FUNCTION_BLOCK DynamicStringBuffer_TEST EXTENDS FB_TestSuite
VAR_INPUT
END_VAR
VAR_OUTPUT
END_VAR
VAR
END_VAR

LogsManyMessagesForManyCycles();

METHOD LogsManyMessagesForManyCycles
VAR_INPUT
END_VAR
VAR
	result: STRING := '';
	expected: STRING := '';
	i: UDINT;
END_VAR

VAR CONSTANT
	CYCLES: UDINT := 30;
	MESSAGES: UDINT := 30;
END_VAR

VAR_INST
	cycleCount: UDINT := 0;
	LogsManyMessagesForManyCyclesLogger: TcLogCore(nBufferSize := 30*30*280); // cycles * messages * (max string length + fifo overhead (estimated))
	logger: TcLog;
END_VAR
TEST('LogsManyMessagesForManyCycles');

LogsManyMessagesForManyCyclesLogger
	.WriteToFile('c:\logs\', 'test.txt')
	.RunLogger();
logger.SetLogger(LogsManyMessagesForManyCyclesLogger);

IF cycleCount < CYCLES THEN
	FOR i:=0 TO MESSAGES DO
		logger
			.AppendString('Cycle: ')
			.AppendString(UDINT_TO_STRING(cycleCount))
			.AppendString(', Message: ')
			.AppendString(UDINT_TO_STRING(i))
			.Error('');	
	END_FOR
END_IF
cycleCount := cycleCount + 1;

// Length of operations (empirically determined):
// file open: 		2 cycles
// pop from fifo: 	1-2 cycle
// write to file: 	2 cylces
// close file:		2 cylces
// => thus for x messages you need 4 * x + 4 cycles

// Catch any occuring error message
IF LEN(LogsManyMessagesForManyCyclesLogger.Error.Info) > 0 THEN
	result := LogsManyMessagesForManyCyclesLogger.Error.Info;
END_IF

IF cycleCount > (CYCLES * MESSAGES * 4 + 10) THEN 
	AssertEquals(Expected := expected,
				 Actual := result,
				 Message := result);
 
	TEST_FINISHED();
END_IF
END_METHOD

END_FUNCTION_BLOCK

(* stored: Version 1.1.0.1, ProductVersion 3.1.4024.11
   POU DynamicStringBuffer_TEST: Id {03045c1a-5281-4fe3-bc16-4d9ce12d6b50}, SpecialFunc None
   Method LogsManyMessagesForManyCycles: Id {e452a053-adba-401f-a1d2-1bba967ad2c0} *)
